(* CoDeSys 2.3.9.31 project: derevo_2014_05_18.pr6 *)
(* Author: Yurko Shybaigolova *)
(* Libraries: TcAdsBC.lb6 5.7.02 12:03:02, STANDARD.LB6 5.6.98 12:03:02 *)

(* Global variable list: main *)
VAR_GLOBAL
	data3floor: ARRAY[0..100] OF BYTE;
	data3floor_prev :ARRAY[0..100] OF BYTE;

	ads_adr1: STRING:='10.0.5.61.1.1';
	ads_adr2: STRING:='10.0.5.62.1.1';
	ads_adr3: STRING:='10.0.5.63.1.1';

	write_ads: ADSWRITE;

	T_out3			AT%MB403:BYTE;


	iHour			AT%MB404:BYTE;
	iMinute			AT%MB405:BYTE;
	lights			AT%MB406:DWORD;

	bDarkOutside		AT%MX400.6:BOOL;
	bT_out_sign		AT%MX400.7:BOOL;

	eib_vidpochynok1 AT %MX500.0:	 BOOL;
	eib_vidpochynok2 AT %MX500.1:	 BOOL;
	eib_veranda AT %MX500.2:	 BOOL;
	eib_veranda_zovn AT %MX500.3:	 BOOL;
	eib_vhid_zovn AT %MX500.4:	 BOOL;
	eib_sauna AT %MX500.5:	 BOOL;
	eib_vhid	AT %MX500.6:	 BOOL;
	eib_kotel AT %MX500.7:	 BOOL;
	eib_korydor AT %MX501.0:	 BOOL;
	eib_sinna AT %MX501.1:	 BOOL;
	eib_hamam AT %MX501.2:	 BOOL;
	eib_kuhnya AT %MX501.3:	 BOOL;
	eib_bassein1	AT %MX501.4:	 BOOL;
	eib_bassein2	AT %MX501.5:	 BOOL;
	eib_spalnya2	AT %MX501.6:	 BOOL;
	eib_terassa AT %MX501.7:	 BOOL;
	eib_dush AT %MX502.0:	 BOOL;
	eib_wc AT %MX502.1:	 BOOL;
	eib_spalnya_verh	AT %MX502.2:	 BOOL;
	eib_spalnya1 AT %MX502.3:	 BOOL;
	eib_spalnya_su AT %MX502.4:	 BOOL;
	eib_garderob AT %MX502.5:	 BOOL;


END_VAR

(* Global variable list: physical *)
(* @GLOBAL_VARIABLE_LIST := TwinCAT_Import *)
(* @PATH := '' *)
VAR_GLOBAL (* DO NOT CHANGE THIS SHEET MANUALLY! *)
	PlcInVar_0	AT %QB128:	USINT;
	PlcInVar_1	AT %QB129:	USINT;
	PlcInVar_2	AT %QB130:	USINT;
	PlcInVar_3	AT %QB131:	USINT;
	PlcInVar_4	AT %QB132:	USINT;
	PlcInVar_5	AT %QB133:	USINT;
	PlcInVar_6	AT %QB134:	USINT;
	PlcInVar_7	AT %QB135:	USINT;
	PlcInVar_8	AT %QB136:	USINT;
	PlcInVar_9	AT %QB137:	USINT;
	PlcInVar_10	AT %QB138:	USINT;
	PlcInVar_11	AT %QB139:	USINT;
	PlcInVar_12	AT %QB140:	USINT;
	PlcInVar_13	AT %QB141:	USINT;
	PlcInVar_14	AT %QB142:	USINT;
	PlcInVar_15	AT %QB143:	USINT;
	PlcOutVar_0	AT %IB128:	USINT;
	PlcOutVar_1	AT %IB129:	USINT;
	PlcOutVar_2	AT %IB130:	USINT;
	PlcOutVar_3	AT %IB131:	USINT;
	PlcOutVar_4	AT %IB132:	USINT;
	PlcOutVar_5	AT %IB133:	USINT;
	PlcOutVar_6	AT %IB134:	USINT;
	PlcOutVar_7	AT %IB135:	USINT;
	PlcOutVar_8	AT %IB136:	USINT;
	PlcOutVar_9	AT %IB137:	USINT;
	PlcOutVar_10	AT %IB138:	USINT;
	PlcOutVar_11	AT %IB139:	USINT;
	PlcOutVar_12	AT %IB140:	USINT;
	PlcOutVar_13	AT %IB141:	USINT;
	PlcOutVar_14	AT %IB142:	USINT;
	PlcOutVar_15	AT %IB143:	USINT;
	term1 AT%QB0:BYTE;
	term2 AT%QB1:BYTE;
	term3 AT%QB2:BYTE;
	term4 AT%QB3:BYTE;
	vidpochynok1	AT %QX0.0:	BOOL;
	vidpochynok2	AT %QX0.1:	BOOL;
	veranda 		AT %QX0.2:	BOOL;
	veranda_zovn	AT %QX0.3:	BOOL;
	vhid_zovn		AT %QX0.4:	BOOL;
	sauna			AT %QX0.5:	BOOL;
	vhid			AT %QX0.6:	BOOL;
(*c8*)kotel			AT %QX0.7:	BOOL;
	korydor			AT %QX1.0:	BOOL;
	sinna			AT %QX1.1:	BOOL;
	hamam			AT %QX1.2:	BOOL;
	kuhnya			AT %QX1.3:	BOOL;
	bassein1		AT %QX1.4:	BOOL;
	bassein2		AT %QX1.5:	BOOL;
	spalnya2		AT %QX1.6:	BOOL;
	terassa			AT %QX1.7:	BOOL;
	dush			AT %QX2.0:	BOOL;
	wc				AT %QX2.1:	BOOL;
	spalnya_verh	AT %QX2.2:	BOOL;
	spalnya1		AT %QX2.3:	BOOL;
	spalnya_su		AT %QX2.4:	BOOL;
	garderob		AT %QX2.5:	BOOL;
	Term_3_KL2408_7_Output	AT %QX2.6:	BOOL;
	Term_3_KL2408_8_Output	AT %QX2.7:	BOOL;

	dush2			AT %QX3.0:	BOOL;
	bassein_lampa	AT %QX3.1:	BOOL;
	Term_4_KL2408_3_Output	AT %QX3.2:	BOOL;
	Term_4_KL2408_4_Output	AT %QX3.3:	BOOL;
	Term_4_KL2408_5_Output	AT %QX3.4:	BOOL;
	Term_4_KL2408_6_Output	AT %QX3.5:	BOOL;
	Term_4_KL2408_7_Output	AT %QX3.6:	BOOL;
	Term_4_KL2408_8_Output	AT %QX3.7:	BOOL;




	sw_vidpochynok1			AT %IX0.0:	BOOL;
	sw_vidpochynok2			AT %IX0.1:	BOOL;
	sw_veranda1				AT %IX0.2:	BOOL;
	sw_veranda2				AT %IX0.3:	BOOL;
	sw_spalnya1				AT %IX0.4:	BOOL;
	sw_spalnya2				AT %IX0.5:	BOOL;
	sw_vhid1			AT %IX0.6:	BOOL;
	sw_vhid2			AT %IX0.7:	BOOL;
	sw_korydor1				AT %IX1.0:	BOOL;
	sw_korydor2				AT %IX1.1:	BOOL;
	sw_vidpochynok_skhody1	AT %IX1.2:	BOOL;
	sw_vidpochynok_skhody2	AT %IX1.3:	BOOL;
	sw_sauna1				AT %IX1.4:	BOOL;
	sw_sauna2				AT %IX1.5:	BOOL;
	sw_bassein1				AT %IX1.6:	BOOL;
	sw_bassein2				AT %IX1.7:	BOOL;
	sw_sauna_vhid2		AT %IX2.0:	BOOL;
	sw_sauna_vhid1		AT %IX2.1:	BOOL;
	sw_sinna1					AT %IX2.2:	BOOL;
	Term_7_KL1408_4_Input	AT %IX2.3:	BOOL;
	sw_spalnya_su				AT %IX2.4:	BOOL;
	sw_garderob				AT %IX2.5:	BOOL;
	sw_kuh1					AT %IX2.6:	BOOL;
	sw_kuh2					AT %IX2.7:	BOOL;
	Term_8_KL1408_1_Input	AT %IX3.0:	BOOL;
	sw_sinna						AT %IX3.1:	BOOL;
	sw_skhody_22					AT %IX3.2:	BOOL;
	sw_skhody_21					AT %IX3.3:	BOOL;
	sw_skhody_12					AT %IX3.4:	BOOL;
	sw_skhody_11					AT %IX3.5:	BOOL;
	sw_hamam					AT %IX3.6:	BOOL;
	sw_spalnya_verh			AT %IX3.7:	BOOL;
	sw_terr1					AT %IX4.0:	BOOL;
	sw_terr2					AT %IX4.1:	BOOL;
	Term_9_KL1408_3_Input	AT %IX4.2:	BOOL;
	Term_9_KL1408_4_Input	AT %IX4.3:	BOOL;
	Term_9_KL1408_5_Input	AT %IX4.4:	BOOL;
	Term_9_KL1408_6_Input	AT %IX4.5:	BOOL;
	Term_9_KL1408_7_Input	AT %IX4.6:	BOOL;
	Term_9_KL1408_8_Input	AT %IX4.7:	BOOL;
END_VAR

(* @OBJECT_END := TwinCAT_Import *)

VAR_GLOBAL
END_VAR

(* POU MAIN, ST *)
PROGRAM MAIN
VAR

	g_veranda				:	SWITCH;
	g_spalnya1				:	SWITCH;
	g_spalnya2				:	SWITCH;
	g_sauna_skhody1			:	SWITCH;
	g_sauna_skhody2			:	SWITCH;
	g_bassein_skhody1		:	SWITCH;
	g_bassein_skhody2		:	SWITCH;
	g_vidpochynok_skhody1	:	SWITCH;
	g_vidpochynok_skhody2	:	SWITCH;
	g_sauna_vhid1				:	SWITCH;
	g_sauna_vhid2				:	SWITCH;
	g_bassein1				:	SWITCH;
	g_bassein2				:	SWITCH;
	g_sauna_skhody2_1		:	SWITCH;
	g_sauna_skhody2_2		:	SWITCH;
	g_sinna					:	SWITCH;
	g_Term_7_KL1408_4_Input	:	SWITCH;
	g_spalnya_su				:	SWITCH;
	g_garderob				:	SWITCH;
	g_kuh1					:	SWITCH;
	g_kuh2					:	SWITCH;

	g_sinna1						:	SWITCH;
	g_skhody_22					:	SWITCH;
	g_skhody_21					:	SWITCH;
	g_skhody_12					:	SWITCH;
	g_skhody_11					:	SWITCH;
	g_hamam					:	SWITCH;

	delay: TIME;
	g_vidpochynok1: SWITCH;
	g_vidpochynok2: SWITCH;
	g_veranda1: SWITCH;
	g_zovn: SWITCH;
	g_korydor: SWITCH;
	g_bassein: SWITCH;
	g_terassa: SWITCH;
	g_vhid: SWITCH;
	g_dush: SWITCH;
	g_wc: SWITCH;
	g_sauna: SWITCH;
	g_vhid_zovn: SWITCH;

	F_polka:F_TRIG;
	R_polka: R_TRIG;

	g_spalnya_verh: SWITCH;


	prev_eib_vidpochynok1 :	 BOOL;
	prev_eib_vidpochynok2 :	 BOOL;
	prev_eib_veranda :	 BOOL;
	prev_eib_veranda_zovn :	 BOOL;
	prev_eib_vhid_zovn :	 BOOL;
	prev_eib_sauna :	 BOOL;
	prev_eib_vhid	:	 BOOL;
	prev_eib_kotel:	 BOOL;
	prev_eib_korydor :	 BOOL;
	prev_eib_sinna :	 BOOL;
	prev_eib_hamam :	 BOOL;
	prev_eib_kuhnya :	 BOOL;
	prev_eib_bassein1	:	 BOOL;
	prev_eib_bassein2	:	 BOOL;
	prev_eib_spalnya2	:	 BOOL;
	prev_eib_terassa :	 BOOL;
	prev_eib_dush :	 BOOL;
	prev_eib_wc :	 BOOL;
	prev_eib_spalnya_verh	:	 BOOL;
	prev_eib_spalnya1 :	 BOOL;
	prev_eib_spalnya_su :	 BOOL;
	prev_eib_garderob :	 BOOL;
END_VAR
delay:=t#1s;
	g_vidpochynok1(IN:=sw_vidpochynok1  XOR sw_vidpochynok_skhody1 XOR sw_skhody_11, SWITCH_DELAY:=delay,Q_SHORT=>vidpochynok1);

IF eib_vidpochynok1=prev_eib_vidpochynok1 THEN
	IF g_vidpochynok1.short THEN vidpochynok1:=NOT vidpochynok1; eib_vidpochynok1:=vidpochynok1; END_IF;
ELSE
	vidpochynok1:=eib_vidpochynok1;
END_IF


	g_vidpochynok2(IN:=sw_vidpochynok2, SWITCH_DELAY:=delay,Q_SHORT=>vidpochynok2);
	g_kuh1	(IN:=sw_kuh1 , SWITCH_DELAY:=delay,Q_SHORT=>kuhnya);
	g_kuh2	(IN:=sw_kuh2, SWITCH_DELAY:=delay(*kuhnya_pidsvitka*));

	g_veranda(IN:=sw_veranda1, SWITCH_DELAY:=delay,Q_SHORT=>veranda);

	g_zovn(IN:=sw_veranda2, SWITCH_DELAY:=delay,Q_SHORT=>veranda_zovn);

	g_spalnya1	(MODE:='short&long',IN:=sw_spalnya1, SWITCH_DELAY:=delay,Q_SHORT=>spalnya1);

	g_spalnya_verh( IN:=sw_spalnya_verh, SWITCH_DELAY:=delay);


F_polka(CLK:=g_spalnya1.Q_LONG XOR g_spalnya_verh.Q_SHORT);
R_polka(CLK:=g_spalnya_verh.Q_SHORT XOR g_spalnya1.Q_LONG );
IF F_polka.Q OR R_polka.Q THEN spalnya_verh:= NOT spalnya_verh; END_IF


	g_spalnya2	(IN:=sw_spalnya2, SWITCH_DELAY:=delay,Q_SHORT=>spalnya2);

	g_bassein(IN:=sw_korydor1 XOR sw_skhody_12, SWITCH_DELAY:=delay,Q_SHORT=>bassein1);
bassein2:=bassein1;

	g_terassa(IN:=sw_vidpochynok_skhody2, SWITCH_DELAY:=delay,Q_SHORT=>terassa);

	g_korydor(IN:= sw_korydor2 XOR  sw_sauna_vhid2 , SWITCH_DELAY:=delay,Q_SHORT=>korydor);

	g_sauna	(IN:=sw_sauna2, SWITCH_DELAY:=delay,Q_SHORT=>sauna);

	g_wc(IN:=sw_bassein1 XOR sw_skhody_21, SWITCH_DELAY:=delay,Q_SHORT=>wc);

	g_dush (IN:=sw_bassein2 XOR sw_skhody_22, SWITCH_DELAY:=delay,Q_SHORT=>dush);

	g_spalnya_su(IN:=sw_spalnya_su, SWITCH_DELAY:=delay,Q_SHORT=>spalnya_su);

	g_garderob	(IN:=sw_garderob, SWITCH_DELAY:=delay,Q_SHORT=>garderob);

	g_sinna(IN:=sw_sinna, SWITCH_DELAY:=delay,Q_SHORT=>sinna);

	g_hamam(IN:=sw_hamam, SWITCH_DELAY:=delay,Q_SHORT=>hamam);

	g_vhid_zovn(IN:=sw_vhid1 ,SWITCH_DELAY:=delay,Q_SHORT=>vhid_zovn);
	g_vhid(IN:=sw_sauna_vhid1 XOR sw_vhid2, SWITCH_DELAY:=delay,Q_SHORT=>vhid);

	prev_eib_vidpochynok1 :=eib_vidpochynok1 ;
	prev_eib_vidpochynok2 :=eib_vidpochynok2 ;
	prev_eib_veranda :=eib_veranda ;
	prev_eib_veranda_zovn :=eib_veranda_zovn ;
	prev_eib_vhid_zovn :=eib_vhid_zovn ;
	prev_eib_sauna :=eib_sauna ;
	prev_eib_vhid:=eib_vhid	;
	prev_eib_kotel:=eib_kotel;
	prev_eib_korydor :=eib_korydor ;
	prev_eib_sinna:=eib_sinna ;
	prev_eib_hamam :=eib_hamam ;
	prev_eib_kuhnya :=eib_kuhnya ;
	prev_eib_bassein1:=eib_bassein1	;
	prev_eib_bassein2:=eib_bassein2;
	prev_eib_spalnya2:=eib_spalnya2;
	prev_eib_terassa:=eib_terassa;
	prev_eib_dush:=eib_dush ;
	prev_eib_wc :=eib_wc ;
	prev_eib_spalnya_verh:=eib_spalnya_verh	;
	prev_eib_spalnya1:=eib_spalnya1 ;
	prev_eib_spalnya_su:=eib_spalnya_su ;
	prev_eib_garderob :=eib_garderob ;

	data3floor[0].0:= vidpochynok1 ;
	data3floor[0].1:= vidpochynok2 ;
	data3floor[0].2:= veranda ;
	data3floor[0].3:= veranda_zovn ;
	data3floor[0].4:= vhid_zovn ;
	data3floor[0].5:= sauna ;
	data3floor[0].6:= vhid	;
	data3floor[0].7:= kotel;
	data3floor[1].0:= korydor ;
	data3floor[1].1:= sinna ;
	data3floor[1].2:= hamam ;
	data3floor[1].3:= kuhnya ;
	data3floor[1].4:= bassein1	;
	data3floor[1].5:= bassein2;
	data3floor[1].6:= spalnya2;
	data3floor[1].7:= terassa;
	data3floor[2].0:= dush ;
	data3floor[2].1:= wc ;
	data3floor[2].2:= spalnya_verh	;
	data3floor[2].3:= spalnya1 ;
	data3floor[2].4:= spalnya_su ;
	data3floor[2].5:= garderob ;



ADS_write;
END_PROGRAM

(* POU Vymykachi/SWITCH, ST *)
FUNCTION_BLOCK SWITCH
VAR_INPUT
	IN:BOOL;
	SWITCH_DELAY:TIME; (*різниця між коротким і довгим натисненням*)
	SHORT_OFF_DELAY, LONG_OFF_DELAY: TIME; (*час затримки вимкнення по короткому та довгому натисненню*)
	MODE:STRING; (*delayed, light, light&vent, short&long, delayed_short&long, *)
	NUMBER_OF_OUTS:INT;
END_VAR
VAR_OUTPUT
	Q_SHORT:BOOL:=FALSE;
	Q_SHORT_D: BOOL;(*вихід для вимкнення із затримкою, вмикається разом із виходом короткого натискання*)
	Q_LONG:BOOL:=FALSE;
	Q_LONG_D:BOOL; (*вихід для вимкнення із затримкою, вмикається разом із виходом довгого натискання*)
END_VAR
VAR
	STAN:BOOL:=FALSE;
	Q_S_fall:F_TRIG; (*ловить задній фронт вихода короткого натискання*)
	Q_L_fall:F_TRIG;(*ловить задній фронт вихода довгого натискання*)
	chas: TIME; (*час доки кнопка натиснена*)

	long: BOOL; (*стає тру, якщо було довге натиснення*)
	short: BOOL; (*стає тру, якщо було коротке натиснення*)
	timer, short_off_delay_timer, long_off_delay_timer: TON; (*таймери: час натискання, час переключення відкладеного виходу по довгому та короткому натисканнях*)
	up: BOOL; (*кнопка натиснена*)

	delay_l, delay_s:BOOL; (*запускати таймери відкладеного вимкнення*)

	turn_off_long: BOOL;
	start_l, start_s:BOOL;
END_VAR
short:=0;
long:=0;
timer(IN:=IN AND STAN, PT:=t#10s);
IF IN AND STAN THEN
	chas:=timer.ET;
	up:=1;
ELSE
up:=0;
END_IF;

IF NOT IN AND NOT STAN THEN
chas:=t#0ms;
END_IF;

IF STAN AND NOT IN THEN
	IF chas <SWITCH_DELAY THEN
		short:=1;
		Q_SHORT:= NOT Q_SHORT;
	END_IF;
	IF chas>=SWITCH_DELAY THEN
		Q_LONG:= NOT Q_LONG;
		long:=1;
	END_IF;
END_IF;

(*затримка вимикання*)
Q_L_fall(CLK:=Q_LONG);
Q_S_fall(CLK:=Q_SHORT);

IF Q_L_FALL.Q THEN
		start_l:=TRUE;
END_IF

IF Q_S_FALL.Q THEN
	start_s:=TRUE;
END_IF

IF MODE='light&vent' THEN
	IF start_s THEN start_l:=start_s; END_IF
END_IF

IF LONG_OFF_DELAY <> t#0ms THEN (*виконувати лише якщо в блок переданий параметр затримки на вимкнення*)

	IF Q_LONG THEN
		Q_LONG_D:=Q_LONG;
	END_IF

	long_off_delay_timer(IN:=start_l, PT:=LONG_OFF_DELAY);

	IF long_off_delay_timer.Q THEN
		Q_LONG_D:=FALSE;
		start_l:=FALSE;
	END_IF

ELSE
	Q_LONG_D:=Q_LONG;
END_IF

IF SHORT_OFF_DELAY <> t#0ms THEN (*виконувати лише якщо в блок переданий параметр затримки на вимкнення*)

	IF Q_SHORT THEN
		Q_SHORT_D:=Q_SHORT;
	END_IF

	short_off_delay_timer(IN:=start_s, PT:=SHORT_OFF_DELAY);

	IF short_off_delay_timer.Q THEN
		Q_SHORT_D:=FALSE;
		start_s:=FALSE;
	END_IF


ELSE
	Q_SHORT_D:=Q_SHORT;
END_IF

IF MODE='delayed' THEN
	Q_LONG:=Q_LONG_D;
	Q_SHORT:=Q_SHORT_D;
END_IF
(*працють лише короткі замикання*)
IF MODE='light' THEN
	Q_SHORT_D:=FALSE;
	Q_LONG:=Q_SHORT;
	Q_LONG_D:=FALSE;
END_IF
(*затримки не працюють*)
IF MODE='short&long' THEN
	Q_SHORT_D:=FALSE;
	Q_LONG_D:=FALSE;
END_IF
(*при вимкненні всього світла вимикати вентилятор і затримкою*)
IF MODE='light&vent' THEN
	IF NOT Q_SHORT AND Q_LONG THEN
		Q_LONG:=Q_LONG_D;
	END_IF
END_IF

STAN := IN;
END_FUNCTION_BLOCK

(* POU ADS_write, ST *)
PROGRAM ADS_write
VAR
	write_timeout: TIME;
	b_write3, b_write2: BOOL;
	write_ads3, write_ads2: ADSWRITE;

	timer3, timer2:TP;
	errorcounter3, errorcounter2, pack_c:CTU ;
	test_word: WORD;
	i,j,i1,j1: INT;
	data_changed: BOOL;
	try_again2, try_again3: BOOL;
	temp: INT;
	SENT2, SENT3:F_TRIG;
	SNT_CNT2, SNT_CNT3:CTU;
	fb_heartbeat_timer: TON;
END_VAR
write_timeout:=t#1s;
fb_heartbeat_timer(in:=NOT fb_heartbeat_timer.Q, pt:=t#10s);

(*3floor*)
FOR i1:=0 TO (SIZEOF(data3floor)-1)-1DO
	IF data3floor[i1]<>data3floor_prev[i1] OR fb_heartbeat_timer.Q  THEN
		b_write3:=TRUE;
		EXIT;
	ELSE
		b_write3:=FALSE;
	END_IF
END_FOR

IF try_again3 AND NOT timer3.Q THEN
	b_write3:=TRUE;
	try_again3:=FALSE;
END_IF


IF write_ads3.BUSY THEN b_write3:=FALSE; END_IF

	write_ads3(
		NETID:=ads_adr3,
		PORT:=801,
		IDXGRP:=16#4020,
		IDXOFFS:=400,
		WRITE:=b_write3,
		TMOUT:=write_timeout,
		LEN:=SIZEOF(data3floor),
		SRCADDR:=ADR(data3floor));

IF write_ads3.ERR AND NOT timer3.Q THEN
	timer3.IN:=TRUE;
	try_again3:=TRUE;
END_IF
timer3(PT:=write_timeout);
timer3.IN:=FALSE;

SENT3(CLK:=write_ads3.BUSY);

IF NOT write_ads3.ERR THEN
	SNT_CNT3(CU:=SENT3.Q);
END_IF

FOR j1:=0 TO (SIZEOF(data3floor)-1)-1 DO
	data3floor_prev[j1]:=data3floor[j1];
END_FOR
END_PROGRAM
